// TIA Portal V16 export
// export: Created 2023-03-29T11:03:47.4642075Z, ExportSetting WithDefaults, DisplayName Totally Integrated Automation Portal, DisplayVersion V16 Update 6, DisplayName TIA Portal Version Control Interface, DisplayVersion V16 Update 2, DisplayName TIA Portal Openness, DisplayVersion V16 Update 6, DisplayName STEP 7 Professional, DisplayVersion V16 Update 6, DisplayName STEP 7 Safety, DisplayVersion V16, DisplayName WinCC Advanced, DisplayVersion V16 Update 6
TYPE "typeModbusMaster"
// stored: IsFailsafeCompliant false
   STRUCT
      req : Bool := FALSE;   // The enable to initiate a Modbus master request
      mbAddr : UInt;   // The station address of the Modbus slave
      mode : USInt := 0;   // Specifies a read, write, or diagnostic operation
      dataAddr : UDInt := 0;   // The Modbus data address
      dataLen : UInt := 0;   // The Modbus data length
      done : Bool := FALSE;   // Boolean indicating completion without error
      busy : Bool := FALSE;   // Boolean indicating operation in progress
      error : Bool := FALSE;   // Boolean indicating completion with error
      status : Word := W#16#0;   // Status or error code of the completed operation
      errorStatus : Word := W#16#0;   // Error code of the faulty operation
   END_STRUCT;
END_TYPE
